FUNCTION_BLOCK FB_BaseState IMPLEMENTS Istate
VAR_INPUT
END_VAR
VAR_OUTPUT
END_VAR
VAR
	_pStation		: REFERENCE TO FB_Station;
	bIsInitalized	: BOOL;
END_VAR

METHOD FB_init : BOOL
VAR_INPUT
	bInitRetains : BOOL; // if TRUE, the retain variables are initialized (warm start / cold start)
	bInCopyCode : BOOL;  // if TRUE, the instance afterwards gets moved into the copy code (online change)
	
	StationPointer 	: POINTER TO FB_Station;
END_VAR
END_METHOD

{warning 'add method implementation '}
METHOD mExecute
END_METHOD

{warning 'add method implementation '}
METHOD mHold
END_METHOD

{warning 'add method implementation '}
METHOD mStart
END_METHOD

{warning 'add method implementation '}
METHOD mStop
END_METHOD

PROPERTY pMessage : STRING
GET
END_GET
END_PROPERTY

{attribute 'monitoring' := 'variable'}
PROPERTY pStation : REFERENCE TO FB_Station;
GET
pStation REF= _pStation;
END_GET
SET
_pStation REF= pStation;
END_SET
END_PROPERTY

END_FUNCTION_BLOCK

(* stored: Version 1.1.0.1, ProductVersion 3.1.4024.9
   POU FB_BaseState: Id {8449a010-d346-45fc-ac07-fe9a1eaecc14}, SpecialFunc None
   Method FB_init: Id {48245767-a5cc-40e5-bb2b-835b6d9e87b5}
   Method mExecute: Id {521ddd78-4d09-4566-9d76-1b16d49db34b}
   Method mHold: Id {42dce020-4531-4286-9dce-1d80dd02d5ff}
   Method mStart: Id {d71d28e7-e340-45af-8af7-3f2d84a5abf3}
   Method mStop: Id {b742d1cb-9d9b-4cd4-b8f4-798551bf5b33}
   Property pMessage: Id {28b93941-4340-432d-941d-6b8d7e8b94db}
   Get Get: Id {8761b569-7439-4d25-b331-54b2cdba8ddb}
   Property pStation: Id {03c903f9-b001-462a-9492-cfae314d5c55}
   Get Get: Id {45337113-012a-481e-a096-a31799ecc47c}
   Set Set: Id {ba781cba-cd4a-4613-b5f6-085a54fdb138} *)
